// TIA Portal V20 export
// export: Created 2026-04-11T06:02:30.6421882Z, ExportSetting WithDefaults, DisplayName Totally Integrated Automation Portal, DisplayVersion V20, DisplayName TIA Portal Openness, DisplayVersion V20, DisplayName TIA Portal Version Control Interface, DisplayVersion V20, DisplayName STEP 7 Professional, DisplayVersion V20, DisplayName STEP 7 Safety, DisplayVersion V20, DisplayName WinCC Basic/Comfort/Advanced, DisplayVersion V20, DisplayName WinCC Unified, DisplayVersion V20
TYPE "udtHMI_Brabender"
// stored: IsFailsafeCompliant false
   STRUCT
      iMode : Int;   // Current mode code
      iErrorCode { ExternalWritable := 'False'} : Int;   // Error code
      rManualFlowSP { S7_SetPoint := 'True'} : Real;   // Flow set point - manual mode
      rAutoFlowSP { ExternalWritable := 'False'} : Real;   // Flow set point - auto mode
      rHLProcess { S7_SetPoint := 'True'} : Real;   // Stop refill level
      rLLProcess { S7_SetPoint := 'True'} : Real;   // Start refill level
      bPB_ResetError : Bool;   // PB Reset errors
      bPB_Start : Bool;   // PB start in manual mode
      bPB_Stop : Bool;   // PB Stop in manual mode
      bPB_RefillStart : Bool;   // PB Refill start in manual mode
      bPB_Gravimetric : Bool;   // PB Change mode to gravimetric
      bPB_Cleanout : Bool;   // PB Change mode to discharge/cleanout (VFD % control)
      bPBEN_ResetError { ExternalWritable := 'False'} : Bool;   // PB reset errors enable
      bPBEN_Start { ExternalWritable := 'False'} : Bool;   // PB start enable
      bPBEN_Stop { ExternalWritable := 'False'} : Bool;   // PB stop enable
      bPBEN_RefillStart { ExternalWritable := 'False'} : Bool;   // PB Refill start enable
      bPBEN_Gravimetric { ExternalWritable := 'False'} : Bool;   // PB Change mode to gravimetric enable
      bPBEN_Cleanout { ExternalWritable := 'False'} : Bool;   // PB Change mode to discharge/cleanout (VFD % control) enable
      bRefillRequest { ExternalWritable := 'False'} : Bool;   // Refilling request
      bRefillInProgress { ExternalWritable := 'False'} : Bool;   // Refill in progress
      bRunRequest { ExternalWritable := 'False'} : Bool;   // Feeder run request
      bRunning { ExternalWritable := 'False'} : Bool;   // Feeder is running
      bStartConditionNotMet { ExternalWritable := 'False'} : Bool;   // Start conditions not met
      bInterlock { ExternalWritable := 'False'} : Bool;   // Interlock is on
      bError { ExternalWritable := 'False'} : Bool;   // Overall error
      bPB_OP1Enable : Bool;
      bPB_BTENable : Bool;
      bPBEN_OP1Enable { ExternalWritable := 'False'} : Bool;
      bPBEN_BTENable { ExternalWritable := 'False'} : Bool;
      OutputData : "udtHMI_Brabender_Output";
      InputData { ExternalWritable := 'False'} : "udtHMI_Brabender_Input";   // Inputs from Brabender Controller
   END_STRUCT;
END_TYPE
